(* CODESYS project xlh_rover_remote_signal_test_00_01.project
   Description: Receives some incoming messages and echoes them with CAN-ID +1
   Company: 3S - Smart Software Solutions GmbH
   Version: 1.0.0.0
   Title: CAN Bus API Example
   Author: 3S - Smart Software Solutions GmbH

Project tree, tasks and I/O mapping:
  xLH_base : CODESYS Control for Raspberry Pi 64 SL, CODESYS, order no. 2302000009, version 4.18.0.0
    application app
      libraries: Standard, 3.5.18.0 (System); Util, 3.5.21.0 (System); VisuDialogs, * (System); Memory, * (3S - Smart Software Solutions GmbH); CmpBitmapPool, * (System); CAN API, 1.0.0.4 (CODESYS); MemoryUtils, * (3S - Smart Software Solutions GmbH); CAA CiA 405, 4.3.0.0 (CODESYS)
      task MAIN_TASK (cyclic, interval 10 ms, priority 1) calls MAIN
      task ENIPScannerIOTask (cyclic, interval t#10ms, priority 0) calls EtherNet_IP_Scanner.IOCycle
      task ENIPScannerServiceTask (cyclic, interval t#20ms, priority 30) calls EtherNet_IP_Scanner.ServiceCycle
      program MAIN [ST]
      trace Trace_Switch_Joystick (task MAIN_TASK): MAIN.byDigOutButton, MAIN.byDigInButton, MAIN.fbReadStatusLoopTime.diValue, MAIN.fbJoystick.fXunfiltered, MAIN.fbJoystick.fYunfiltered, MAIN.fbJoystick.fY, MAIN.fbJoystick.fX, MAIN.iDebugRead, MAIN.iDebugWrite
      function block FB_KALMAN_FILTER [ST]: reset
      function block FB_JOYSTICK [ST]
      Symbols
    SoftMotion General Axis Pool
      a_axis : SM_Drive_PosControl, CODESYS, order no. 1805, version 4.18.0.0
          settings: wDriveID = 4; dwRatioTechUnitsDenom = 101846; iRatioTechUnitsNum = -125; eRampType = 1; fSWMaxVelocity = 50; fSWMaxAcceleration = 100; fSWMaxDeceleration = 100; fSWMaxJerk = 1000; fSWLimitNegative = -1000.0; ScalingIncs = 814768; ScalingUnits = 1000; InvertDirection = TRUE; IsLinearMotor = TRUE; MaximumOutputVelocityInt = 40738; MinimumOutputVelocityInt = -40738; Kp = 0.05; MaxFollowingError = 5.0; EnableFollowingErrorCheck = TRUE; DeadTime = 3.0
      x_axis : SM_Drive_PosControl, CODESYS, order no. 1805, version 4.18.0.0
          settings: dwRatioTechUnitsDenom = 101846; iRatioTechUnitsNum = 125; eRampType = 1; fSWMaxVelocity = 50; fSWMaxAcceleration = 100; fSWMaxDeceleration = 100; fSWMaxJerk = 1000; fSWLimitNegative = -1000; ScalingIncs = 814768; ScalingUnits = 1000; IsLinearMotor = TRUE; MaximumOutputVelocityInt = 40738; MinimumOutputVelocityInt = -40738; Kp = 0.05; MaxFollowingError = 5.0; EnableFollowingErrorCheck = TRUE; DeadTime = 3.0
      y_axis : SM_Drive_PosControl, CODESYS, order no. 1805, version 4.18.0.0
          settings: wDriveID = 2; dwRatioTechUnitsDenom = 101846; iRatioTechUnitsNum = 125; eRampType = 1; fSWMaxVelocity = 50; fSWMaxAcceleration = 100; fSWMaxDeceleration = 100; fSWMaxJerk = 1000; fSWLimitNegative = -1000; ScalingIncs = 814768; ScalingUnits = 1000; IsLinearMotor = TRUE; MaximumOutputVelocityInt = 40738; MinimumOutputVelocityInt = -40738; Kp = 0.05; MaxFollowingError = 5.0; EnableFollowingErrorCheck = TRUE; DeadTime = 3.0
      z_axis : SM_Drive_PosControl, CODESYS, order no. 1805, version 4.18.0.0
          settings: wDriveID = 3; dwRatioTechUnitsDenom = 101846; iRatioTechUnitsNum = 125; eRampType = 1; fSWMaxVelocity = 50; fSWMaxAcceleration = 100; fSWMaxDeceleration = 100; fSWMaxJerk = 1000; fSWLimitNegative = -1000; ScalingIncs = 814768; ScalingUnits = 1000; IsLinearMotor = TRUE; MaximumOutputVelocityInt = 40738; MinimumOutputVelocityInt = -40738; Kp = 0.05; MaxFollowingError = 5.0; EnableFollowingErrorCheck = TRUE; DeadTime = 3.0
    GPIOs_A_B : GPIOs B+/Pi2, CODESYS, version 4.15.0.0
        unmapped channels: digital inputs (GPIO0..GPIO31), digital outputs (GPIO0..GPIO31)
    Onewire
    Camera device
      <Leer>
    SPI
    I²C
    CANbus : CANbus, CODESYS, version 4.3.0.0
        settings: Baudrate = 1000 kbit/s
      CANopen_Manager : CANopen_Manager, CODESYS, version 4.3.0.0
          settings: ConfigVersion = 50659584
        xlh_digital_switch_button_led_joystick : xlh_digital_switch_button_led_joystick, xemax ag, order no. 0, version Revision=16#00000001, FileVersion=1.0
            settings: NODEIDSAVED = 1; SDO Timeout = 1000000; PDO_Autoconfig = FALSE; EXPERTSETTINGS = FALSE; PDO 16#1400.COBID = 16#00000201; Process by CANopenManager = TRUE; PDO 16#1800.COBID = 16#00000181; Process by CANopenManager = TRUE; Leds Button.Subindex = 16#01; Leds Switch.Subindex = 16#01; Digital Inputs Button.Subindex = 16#01; Digital Inputs Switch.Subindex = 16#01; Joystick X.Subindex = 16#01; Joystick Y.Subindex = 16#02; Joystick Button.Subindex = 16#03; SDO List.Set COB-ID sync.Index = 16#1005; SDO List.Set COB-ID sync.Subindex = 16#00; SDO List.Set COB-ID sync.Value = 16#00000080; SDO List.Set COB-ID sync.Size = 32; SDO List.Set COB-ID sync.AbortIfError = FALSE; SDO List.Set COB-ID sync.JumpToLine = FALSE; SDO List.Set COB-ID sync.Line = 0; SDO List.Set communication cycle period.Index = 16#1006; SDO List.Set communication cycle period.Subindex = 16#00; SDO List.Set communication cycle period.Value = 16#00000000; SDO List.Set communication cycle period.Size = 32; SDO List.Set communication cycle period.AbortIfError = FALSE; SDO List.Set communication cycle period.JumpToLine = FALSE; SDO List.Set communication cycle period.Line = 0; SDO List.Set Guardtime.Index = 16#100C; SDO List.Set Guardtime.Subindex = 16#00; SDO List.Set Guardtime.Value = 16#000000C8; SDO List.Set Guardtime.Size = 16; SDO List.Set Guardtime.AbortIfError = FALSE; SDO List.Set Guardtime.JumpToLine = FALSE; SDO List.Set Guardtime.Line = 0; SDO List.Set Lifetime.Index = 16#100D; SDO List.Set Lifetime.Subindex = 16#00; SDO List.Set Lifetime.Value = 16#00000003; SDO List.Set Lifetime.Size = 8;
              SDO List.Set Lifetime.AbortIfError = FALSE; SDO List.Set Lifetime.JumpToLine = FALSE; SDO List.Set Lifetime.Line = 0; SDO List.Set Heartbeat Consumer.Index = 16#1016; SDO List.Set Heartbeat Consumer.Subindex = 16#01; SDO List.Set Heartbeat Consumer.Value = 0; SDO List.Set Heartbeat Consumer.Size = 32; SDO List.Set Heartbeat Consumer.AbortIfError = FALSE; SDO List.Set Heartbeat Consumer.JumpToLine = FALSE; SDO List.Set Heartbeat Consumer.Line = 0; SDO List.Disable PDO.Index = 16#1400; SDO List.Disable PDO.Subindex = 16#01; SDO List.Disable PDO.Value = 16#80000201; SDO List.Disable PDO.Size = 32; SDO List.Disable PDO.AbortIfError = FALSE; SDO List.Disable PDO.JumpToLine = FALSE; SDO List.Disable PDO.Line = 0; SDO List.Set transmission type.Index = 16#1400; SDO List.Set transmission type.Subindex = 16#02; SDO List.Set transmission type.Value = 16#FF; SDO List.Set transmission type.Size = 8; SDO List.Set transmission type.AbortIfError = FALSE; SDO List.Set transmission type.JumpToLine = FALSE; SDO List.Set transmission type.Line = 0; SDO List.Set and enable COB-ID.Index = 16#1400; SDO List.Set and enable COB-ID.Subindex = 16#01; SDO List.Set and enable COB-ID.Value = 16#00000201; SDO List.Set and enable COB-ID.Size = 32; SDO List.Set and enable COB-ID.AbortIfError = FALSE; SDO List.Set and enable COB-ID.JumpToLine = FALSE; SDO List.Set and enable COB-ID.Line = 0; SDO List.Disable PDO.Index = 16#1800; SDO List.Disable PDO.Subindex = 16#01; SDO List.Disable PDO.Value = 16#80000181; SDO List.Disable PDO.Size = 32; SDO List.Disable PDO.AbortIfError = FALSE; SDO List.Disable PDO.JumpToLine = FALSE; SDO List.Disable PDO.Line = 0; SDO List.Set transmission type.Index = 16#1800; SDO List.Set transmission type.Subindex = 16#02;
              SDO List.Set transmission type.Value = 16#FF; SDO List.Set transmission type.Size = 8; SDO List.Set transmission type.AbortIfError = FALSE; SDO List.Set transmission type.JumpToLine = FALSE; SDO List.Set transmission type.Line = 0; SDO List.Set inhibit time.Index = 16#1800; SDO List.Set inhibit time.Subindex = 16#03; SDO List.Set inhibit time.Value = 16#0000; SDO List.Set inhibit time.Size = 16; SDO List.Set inhibit time.AbortIfError = FALSE; SDO List.Set inhibit time.JumpToLine = FALSE; SDO List.Set inhibit time.Line = 0; SDO List.Set event time.Index = 16#1800; SDO List.Set event time.Subindex = 16#05; SDO List.Set event time.Value = 16#0000; SDO List.Set event time.Size = 16; SDO List.Set event time.AbortIfError = FALSE; SDO List.Set event time.JumpToLine = FALSE; SDO List.Set event time.Line = 0; SDO List.Set and enable COB-ID.Index = 16#1800; SDO List.Set and enable COB-ID.Subindex = 16#01; SDO List.Set and enable COB-ID.Value = 16#00000181; SDO List.Set and enable COB-ID.Size = 32; SDO List.Set and enable COB-ID.AbortIfError = FALSE; SDO List.Set and enable COB-ID.JumpToLine = FALSE; SDO List.Set and enable COB-ID.Line = 0; ConfigVersion = 50659584
            output app.MAIN.byDigOutButton : USINT  // Leds Button
            output app.MAIN.byDigOutSwitch : USINT  // Leds Switch
            input  app.MAIN.byDigInButton : USINT  // Digital Inputs Button
            input  app.MAIN.byDigInSwitch : USINT  // Digital Inputs Switch
            input  app.MAIN.usJoystickX : USINT  // Joystick X
            input  app.MAIN.usJoystickY : USINT  // Joystick Y
            input  app.MAIN.bJoystickButton : BOOL  // Joystick Button.Bit0
            unmapped channels: Joystick Button
    Ethernet : Ethernet, CODESYS, version 4.2.0.0
        settings: IPAddress = [192,168,1,168]; SubnetMask = [255,255,255,0]; GatewayAddress = [192,168,1,1]; MACAddress = [16#2C,16#CF,16#67,16#BD,16#46,16#37]; NetworkInterfaceName = 'wlan0'; NetworkInterfaceName = "wlan0"; SaveCommunicationSettings = FALSE; IPAddress = [192,168,0,2]; SubnetMask = [255,255,255,0]; GatewayAddress = [0,0,0,0]
      EtherNet_IP_Scanner : EtherNet/IP Scanner, CODESYS, order no. 1, version 4.8.0.0
          settings: IPAddress = [16#C0,16#A8,16#00,16#01]; SubnetMask = [16#00,16#00,16#00,16#00]; GatewayAddress = [16#00,16#00,16#00,16#00]; TCPFlags = 1; Options.Auto-Reestablish Connections = True; Options.Enable QoS = False
        xlh_rover_signal_test : xlh_rover_signal_test, CODESYS, version Major Revision=16#2, Minor Revision = 16#1
            settings: INITIALIZED = TRUE; IP address of Target = [16#C0,16#A8,16#01,16#BD]; Keying.Check Minor Revision = FALSE; RequiredConfigVersion = 50660864; Number of Connections = 1; Connection Settings.Requested packet intervall = 5000 µs; Connection Settings.Connection Timeout Multiplier = 3; Connection Settings.OT Connection Parameters = 17432; Connection Settings.TO Connection Parameters = 17412; Connection Settings.Transport Type = 17; Connection Settings.Transmission inhibit time Scanner = 5000 µs; Connection Settings.Connection Flags = 1056; Connection Settings.Connection Path Size = 8; Connection Settings.Config#2 Size = 2; Connection Settings.Large OT Connection Parameters = 1140850712; Connection Settings.Large TO Connection Parameters = 1140850692; Configuration Data = [16#00,16#00]; Heartbeat Multiplier = 1; byLedSwitch.ReadOnly = False; byLedSwitch.BitSize = 8; byLedSwitch.DataSize = 1; byLedButton.ReadOnly = False; byLedButton.BitSize = 8; byLedButton.DataSize = 1; fJoystickXnorm.ReadOnly = False; fJoystickXnorm.BitSize = 64; fJoystickXnorm.DataSize = 8; fJoystickYnorm.ReadOnly = False; fJoystickYnorm.BitSize = 64; fJoystickYnorm.DataSize = 8; bySwitch.ReadOnly = False; bySwitch.BitSize = 8; bySwitch.DataSize = 1; byButton.ReadOnly = False; byButton.BitSize = 8; byButton.DataSize = 1; byLedSwitch.Name = 'byLedSwitch'; byLedSwitch.HelpString = ''; byLedSwitch.ReadOnly = False; byLedSwitch.BitSize = 8;
              byLedSwitch.DataSize = 1; byLedSwitch.DataType = 'BYTE'; byLedButton.Name = 'byLedButton'; byLedButton.HelpString = ''; byLedButton.ReadOnly = False; byLedButton.BitSize = 8; byLedButton.DataSize = 1; byLedButton.DataType = 'BYTE'; fJoystickXnorm.Name = 'fJoystickXnorm'; fJoystickXnorm.HelpString = ''; fJoystickXnorm.ReadOnly = False; fJoystickXnorm.BitSize = 64; fJoystickXnorm.DataSize = 8; fJoystickXnorm.DataType = 'LREAL'; fJoystickYnorm.Name = 'fJoystickYnorm'; fJoystickYnorm.HelpString = ''; fJoystickYnorm.ReadOnly = False; fJoystickYnorm.BitSize = 64; fJoystickYnorm.DataSize = 8; fJoystickYnorm.DataType = 'LREAL'; bySwitch.Name = 'bySwitch'; bySwitch.HelpString = ''; bySwitch.ReadOnly = False; bySwitch.BitSize = 8; bySwitch.DataSize = 1; bySwitch.DataType = 'BYTE'; byButton.Name = 'byButton'; byButton.HelpString = ''; byButton.ReadOnly = False; byButton.BitSize = 8; byButton.DataSize = 1; byButton.DataType = 'BYTE'; ConfigVersion = 50660864
            input  app.MAIN.byLedSwitch : BYTE  // byLedSwitch
            input  app.MAIN.byLedButton : BYTE  // byLedButton
            output app.MAIN.fJoystickXnorm : LREAL  // fJoystickXnorm
            output app.MAIN.fJoystickYnorm : LREAL  // fJoystickYnorm
            output app.MAIN.bySwitch : BYTE  // bySwitch
            output app.MAIN.byButton : BYTE  // byButton
  libraries: VisuSymbols, 4.5.0.0 (System); DepictorBase, 1.2.0.0 (CODESYS)
  text list GlobalTextList
  5ce3da45-db07-42e7-a21c-a00fff4ed8f6|C:\Users\phe\Downloads\Musterloesung_FUP.PNG
*)

// xLH_base/app/MAIN
PROGRAM MAIN
VAR_INPUT
	// Ethernet IP
	byLedSwitch: BYTE;
	byLedButton: BYTE;
	iDebugRead: INT;
END_VAR
VAR_OUTPUT
	// Ethernet IP
	fJoystickXnorm: LREAL;
	fJoystickYnorm: LREAL;
	bySwitch: BYTE;
	byButton: BYTE;
	iDebugWrite: INT;
END_VAR
VAR
	byDigInSwitch: USINT;
	byDigOutSwitch: USINT;
	byDigInButton: USINT;
	byDigOutButton: USINT;
	usJoystickX: USINT;
	usJoystickY: USINT;
	bJoystickButton: BOOL;
	byDummy: USINT;
	uiDummy: UINT;
	udiDummy: UDINT;
	fDummy: LREAL;
	
	fbJoystick: FB_JOYSTICK;
	bDummy: BOOL;
	iDummy: INT;
END_VAR

byDummy := byDigInButton;
//byDigOutButton := byDigOutButton + 1;

byDummy := byDigInSwitch;
//byDigOutSwitch := byDigInSwitch OR byDigInButton;

byDummy := usJoystickX;
byDummy := usJoystickY;
bDummy := bJoystickButton;
fbJoystick(
	usX:=usJoystickX,
	usY:=usJoystickY,
	fOffsetZeroX:=136.0,
	fOffsetZeroY:=119.0,
	fDeadbandZero:=15.0);
fDummy := fbJoystick.fX;
fDummy := fbJoystick.fY;
fDummy := fbJoystick.fXnorm;
fDummy := fbJoystick.fYnorm;

// Ethernet IP
fJoystickXnorm := fbJoystick.fXnorm;
fJoystickYnorm := fbJoystick.fYnorm;
bySwitch := byDigInSwitch;
byButton := byDigInButton;
iDummy := iDebugRead;

byDigOutSwitch := byLedSwitch;
byDigOutButton := byLedButton;
iDebugWrite := iDebugRead;// Performancetester

END_PROGRAM

// xLH_base/app/FB_JOYSTICK
FUNCTION_BLOCK FB_JOYSTICK
VAR_INPUT
	usX: UsINT;
	usY: USINT;
	fOffsetZeroX: LREAL := 127.0;
	fOffsetZeroY: LREAL := 127.0;
	fDeadbandZero: LREAL := 5.0;
	fR: LREAL := 25.0;
	fQ: LREAL := 1.0;
END_VAR
VAR_OUTPUT
	fX: LREAL;
	fY: LREAL;
	fXunfiltered: LREAL;
	fYunfiltered: LREAL;
	fXnorm: LREAL;
	fYnorm: LREAL;
END_VAR
VAR
	fbFilterX: FB_KALMAN_FILTER;
	fbFilterY: FB_KALMAN_FILTER;
END_VAR

fXunfiltered := TO_LREAL(usX) - fOffsetZeroX;
IF ABS(fXunfiltered) < fDeadbandZero THEN
	fXunfiltered := 0.0;
END_IF

fYunfiltered := TO_LREAL(usY) - fOffsetZeroY;
IF ABS(fYunfiltered) < fDeadbandZero THEN
	fYunfiltered := 0.0;
END_IF

fbFilterX(fX:=fXunfiltered, fR:=fR, fQ:=fQ, fY=>fX);
fbFilterY(fX:=fYunfiltered, fR:=fR, fQ:=fQ, fY=>fY);

fXnorm := LIMIT(-1.0, fX/115.0, 1.0);
fYnorm := LIMIT(-1.0, fY/115.0, 1.0);

END_FUNCTION_BLOCK

// xLH_base/app/FB_KALMAN_FILTER
FUNCTION_BLOCK PUBLIC FB_KALMAN_FILTER
VAR_INPUT
	fX: LREAL;
	fQ: LREAL;
	fR: LREAL;
	bReset: BOOL;
END_VAR
VAR_OUTPUT
	fY: LREAL;
END_VAR
VAR 
	X_hat: LREAL;
	X_hat_min: LREAL;
	poise: LREAL;
	Pmin: LREAL;
	K: LREAL;
	fAvoidZero: LREAL := 0.001;
END_VAR

IF bReset THEN
	reset();
END_IF

K := Pmin/MAX((Pmin + fR), fAvoidZero);
X_hat := X_hat_min + K*(fX - X_hat_min);
poise := (1 - K)*Pmin;
Pmin := poise + fQ;
X_hat_min := X_hat;
fY := X_hat;

ACTION reset:
X_hat := 0.0;
X_hat_min := 0.0;
poise := 0.0;
Pmin := 0.0;
K := 0.0;
fY := 0.0;
END_ACTION

END_FUNCTION_BLOCK
